PROGRAM UnitTests
VAR
	fbTestRound		: Fb_TestRound;
	fbTestSplit		: FB_TestSplit;
END_VAR

TcUnit.RUN();

END_PROGRAM

(* stored: Version 1.1.0.1, ProductVersion 3.1.4024.9
   POU UnitTests: Id {4c031c1b-3750-4044-bc97-31973c09b395}, SpecialFunc None *)
